TYPE ST_XBox_Controller_State_Bits :
STRUCT
	xConnected  		: BIT;
	{attribute 'hide'}
	xFiller1 			: BIT;
	{attribute 'hide'}
	xFiller2			: BIT;
	{attribute 'hide'}
	xFiller3			: BIT;
	{attribute 'hide'}
	xFiller4			: BIT;
	{attribute 'hide'}
	xFiller5			: BIT;
	{attribute 'hide'}
	xFiller6			: BIT;
	{attribute 'hide'}
	xFiller7			: BIT;
	{attribute 'hide'}
	xFiller8			: BIT;
	{attribute 'hide'}
	xFiller9			: BIT;
	{attribute 'hide'}
	xFiller10			: BIT;
	{attribute 'hide'}
	xFiller11			: BIT;
	{attribute 'hide'}
	xFiller12			: BIT;
	{attribute 'hide'}
	xFiller13			: BIT;
	{attribute 'hide'}
	xFiller14			: BIT;
	{attribute 'hide'}
	xFiller15			: BIT;
END_STRUCT
END_TYPE

(* stored: Version 1.1.0.1, ProductVersion 3.1.4024.11
   DUT ST_XBox_Controller_State_Bits: Id {ebb1c573-1dde-4789-b17e-74cabd58c005} *)
